// TwinCAT 3 PLC project ModbusRTU
// ProgramVersion: 3.1.4024.0
// libraries:
//   Tc2_ModbusRTU, * (Beckhoff Automation GmbH)
//   Tc2_Standard, * (Beckhoff Automation GmbH)
//   Tc2_System, * (Beckhoff Automation GmbH)
//   Tc3_Module, * (Beckhoff Automation GmbH)
// project tree:
//   / PlcTask.TcTTO
//   POUs/ FB_Loadcells.TcPOU, FB_Modbus.TcPOU, MAIN.TcPOU
// real-time tasks:
//   TASK PlcTask: cycle T#10ms, priority 20, ADS port 350
// I/O:
//   DEVICE Device 1 (EtherCAT), AmsNetId 192.168.56.1.2.1
//     Term 1 (EK1100) [EK1100 EtherCAT Coupler (2A E-Bus)]
//       Term 2 (EL6021) [EL6021 Interface (RS422/485)]
// variable links:
//   ModbusRTU Instance <-> Device 1 (EtherCAT)/Term 1 (EK1100)/Term 2 (EL6021)
//     PlcTask Inputs/MAIN.Loadcells.Modbus.Master.InData/D[{0..21}] <-> COM TxPDO-Map Inputs/Data In {0..21}  (22 links)
//     PlcTask Inputs/MAIN.Loadcells.Modbus.Master.InData/Status <-> COM TxPDO-Map Inputs/Status
//     PlcTask Outputs/MAIN.Loadcells.Modbus.Master.OutData/Ctrl <-> COM RxPDO-Map Outputs/Ctrl
//     PlcTask Outputs/MAIN.Loadcells.Modbus.Master.OutData/D[{0..21}] <-> COM RxPDO-Map Outputs/Data Out {0..21}  (22 links)

CONFIGURATION ModbusRTU
    RESOURCE PLC ON TwinCAT3
        TASK PlcTask(INTERVAL := T#10ms, PRIORITY := 20);
        PROGRAM MAIN WITH PlcTask : MAIN;
    END_RESOURCE
END_CONFIGURATION

// ---- POUs/MAIN.TcPOU
PROGRAM MAIN
VAR
	Loadcells			: FB_Loadcells(ModbusAddresses:= LoadcellAddresses, ReadPeriod:= T#1s);
	LoadsInKg			: ARRAY[1..MAX_LOADCELLS] OF INT; //loads on loadcells
	LoadcellFaults		: ARRAY[1..MAX_LOADCELLS] OF BOOL; //faults on reading loadcells
END_VAR
VAR CONSTANT
	MAX_LOADCELLS		: UINT:= 10;
	LoadcellAddresses	: ARRAY[1..MAX_LOADCELLS] OF BYTE:= [1,2,3,4,0]; //must end with 0
END_VAR

Loadcells.Cyclic(LoadsInKg:= LoadsInKg, Faults:= LoadcellFaults);

END_PROGRAM

// ---- POUs/FB_Loadcells.TcPOU
{attribute 'no_explicit_call' := 'do not call FB_Loadcells directly'}
FUNCTION_BLOCK PUBLIC FB_Loadcells
VAR
	Modbus			: FB_Modbus;
	ModbusAddresses	: ARRAY[1..MAX_LOADCELLS] OF BYTE; //addresses of loadcells to read, end with a 0 address
	ModbusErrors	: ARRAY[1..MAX_LOADCELLS] OF MODBUS_ERRORS; //keep track of errors
	_numLoadcells	: UINT; //number of actual addresses to read from above array
	ReadPeriod		: TIME; //poll the loadcells with this period if we can, else just go as fast as we can
	LoadcellsState	: (Idle,ReadLoadcell,WaitForResult,GetReadyForNextRead,Error);
	_cursor			: UINT;
	ReadPeriodTimer	: TON;
END_VAR
VAR CONSTANT
	MAX_LOADCELLS	: UINT:= 10;
END_VAR

METHOD PUBLIC Cyclic
VAR_IN_OUT
	LoadsInKg		: ARRAY[1..MAX_LOADCELLS] OF UINT; //loads on loadcells
END_VAR
VAR
	_allgood		: BOOL;
	_busy			: BOOL;
	_errorID		: MODBUS_ERRORS;
END_VAR
VAR_INST
	kg				: WORD;
	InitDone		: BOOL:= FALSE;
END_VAR
IF NumLoadcells = 0 THEN
	RETURN;
END_IF

IF NOT InitDone THEN
	Init();
	InitDone:= TRUE;
END_IF

ReadPeriodTimer(IN:= TRUE, PT:= ReadPeriod);

//Modbus.Cyclic();

CASE LoadcellsState OF
	Idle:
		//

	ReadLoadcell:
		Modbus.ReadHoldingRegisters(UnitID:= ModbusAddresses[_cursor],
										Quantity:= 1, //only interested in a single register
										MBAddr:= 0, //the first in-fact (400001 is current load in kg)
										Timeout:= T#1S,
										StartedNewRead => _allgood);
		IF _allgood THEN
			LoadcellsState:= WaitForResult;
		END_IF

	WaitForResult:
		Modbus.Cyclic(Busy => _busy, ErrorID => _errorID, FirstRegister => kg);
		IF NOT _busy THEN
			LoadsInKg[_cursor]:= WORD_TO_UINT(kg);
			ModbusErrors[_cursor]:= _errorID;
			LoadcellsState:= GetReadyForNextRead;
		END_IF

	GetReadyForNextRead:
		IF _cursor < NumLoadcells THEN
			_cursor:= _cursor + 1;
			LoadcellsState:= ReadLoadcell;
		ELSE
			IF ReadPeriodTimer.Q THEN
				_cursor:= 1;
				ReadPeriodTimer(IN:= FALSE);
				LoadcellsState:= ReadLoadcell;
			END_IF
		END_IF
END_CASE
END_METHOD

METHOD FB_init : BOOL
VAR_INPUT
	bInitRetains	: BOOL; // if TRUE, the retain variables are initialized (warm start / cold start)
	bInCopyCode		: BOOL;  // if TRUE, the instance afterwards gets moved into the copy code (online change)
	ModbusAddresses	: ARRAY[1..MAX_LOADCELLS] OF BYTE; //array of modbus addresses to read, end with a 0 address
	ReadPeriod		: TIME; //poll the loadcells every ReadPeriod, if this is too short then poll as fast as we can
END_VAR
VAR
	i				: UINT;
	FoundEnd		: BOOL:= FALSE;
END_VAR
THIS^.ModbusAddresses:= ModbusAddresses;
THIS^.ReadPeriod:= ReadPeriod;
FOR i:= 1 TO MAX_LOADCELLS DO
	IF THIS^.ModbusAddresses[i] = 0 THEN
		_numLoadcells:= i - 1;
		FoundEnd:= TRUE;
		EXIT;
	END_IF
END_FOR
IF NOT FoundEnd THEN
	_numLoadcells:= MAX_LOADCELLS;
END_IF
END_METHOD

METHOD PRIVATE Init
VAR_INPUT
END_VAR
LoadcellsState:= ReadLoadcell;
_cursor:= 1;
ReadPeriodTimer(IN:= FALSE);
END_METHOD

PROPERTY PUBLIC NumLoadcells : UINT
GET
NumLoadcells:= _numLoadcells;
END_GET
END_PROPERTY

END_FUNCTION_BLOCK

// ---- POUs/FB_Modbus.TcPOU
{attribute 'no_explicit_call' := 'do not call FB_Modbus directly'}
FUNCTION_BLOCK PUBLIC FB_Modbus
VAR
	Master				: ModbusRtuMaster_KL6x22B;
	ModbusData			: ARRAY[1..DATA_SIZE] OF WORD;
	ModbusState			: (Idle,HR_WaitForResult,HR_Done,HR_Error);
	CyclicBusy			: BOOL; //TRUE if Cyclic is busy and not ready for a new call to Master to commence
	InitDone			: BOOL:= FALSE;
	
	//read holding registers specific
	HR_Quantity			: WORD;
END_VAR
VAR CONSTANT
	DATA_SIZE			: INT:= 20; //maximum size of data we can deal with
	FIRST_REGISTER		: INT:= 1;
END_VAR

METHOD PUBLIC Cyclic
VAR_OUTPUT
	Busy			: BOOL;
	Error			: BOOL;
	ErrorID			: MODBUS_ERRORS;
	FirstRegister	: WORD; //the first register from the read - useful if caller is only interested in a single register
	AllRegisters	: ARRAY[1..DATA_SIZE] OF WORD; //if more than 1 register is asked for, then the results of the read is copied to here
END_VAR
Master.ReadRegs(Execute:= FALSE);

CASE ModbusState OF
	Idle:
		CyclicBusy:= FALSE;

	//read holding registers
	HR_WaitForResult:
		IF NOT MasterBusy AND NOT MasterError THEN
			ModbusState:= HR_Done;
		ELSIF MasterError THEN
			ModbusState:= HR_Error;
		END_IF
		CyclicBusy:= TRUE;

	HR_Done:
		FirstRegister:= ModbusData[1];
		IF HR_Quantity > 1 THEN
			//only do array copy if we need more than one register
			AllRegisters:= ModbusData;
		END_IF
		ModbusState:= Idle;
		CyclicBusy:= FALSE;

	HR_Error:
		FirstRegister:= 0;
		MEMSET(ADR(AllRegisters), 0, SIZEOF(AllRegisters));
		ModbusState:= Idle;
		CyclicBusy:= FALSE;
END_CASE

Busy:= CyclicBusy;
Error:= MasterError;
ErrorID:= MasterErrorID;
END_METHOD

METHOD PRIVATE Init
IF NOT InitDone THEN
	ModbusState:= Idle;
	CyclicBusy:= FALSE;
	InitDone:= TRUE;
END_IF
END_METHOD

PROPERTY PRIVATE MasterBusy : BOOL
GET
MasterBusy:= Master.BUSY;
END_GET
END_PROPERTY

PROPERTY PRIVATE MasterError : BOOL
GET
MasterError:= Master.Error;
END_GET
END_PROPERTY

PROPERTY PRIVATE MasterErrorID : MODBUS_ERRORS
GET
MasterErrorID:= Master.ErrorId;
END_GET
END_PROPERTY

METHOD PUBLIC ReadHoldingRegisters : BOOL
//start a new read of holding registers
VAR_INPUT
	UnitID			: BYTE; //Modbus station address [1..247]
	Quantity		: WORD; //number of data words to read
	MBAddr			: WORD; //Modbus data address to start reading from
	Timeout			: TIME; //wait for up to this long to get result from slave
END_VAR

VAR_OUTPUT
	StartedNewRead	: BOOL;
END_VAR
Init();
IF MasterBusy THEN
	//can't start a new read if we are busy doing something else
	StartedNewRead:= FALSE;
ELSE
	//we don't do any validity checks as the Master FB does those
	Master.ReadRegs(
		UnitID:= UnitID,
		Quantity:= Quantity,
		MBAddr:= MBAddr,
		cbLength:= SIZEOF(ModbusData),
		pMemoryAddr:= ADR(ModbusData),
		Execute:= TRUE,
		Timeout:= Timeout);
	HR_Quantity:= Quantity;
	StartedNewRead:= TRUE;
	ModbusState:= HR_WaitForResult;
END_IF
END_METHOD

END_FUNCTION_BLOCK
